# B&R Automation Studio project VPAKRT
Automation Studio 4.0.17.85 SP

## Configuration Simulation

CPU , AutomationRuntime D4.05

### Task classes (Cpu.sw)
```
Cyclic#1 (cycle 2000 us, tolerance 0 us):
  Reject <- Reject.prg
  main <- main.prg
  Entry <- Entry.prg
  CheckRejec <- CheckReject.prg
  Accumulato <- Accumulator.prg
  Camera1 <- Camera1.prg
  Printer <- Printer.prg
  Conveyor <- Conveyor.prg
Cyclic#4 (cycle 1000000 us, tolerance 10000000 us):
  SerialCode <- SerialCodes.prg
  IHM <- IHM.prg
VcDataObjects: Visu <- Visu.dob
Binaries: sysconf, ashwd, asfw, iomap, arconfig
Libraries: CPP, standard, AsHttp, runtime, AsIecCon, astime, FileIO, sys_lib
```

### Hardware
```
PC_any : PC_any v1.1.0.0 (OrderNumber=PC)
  Connector IF3:
    Vnc1
    VncVcObjectName1 = Visu
    VncKeyMappingFile1 = VC\PS2-Keyboard.dis
  SystemTick = 2000
  TaskClassIdleTime = 2000
  Cyclic1Duration = 2000
  Cyclic1Tolerance = 0
  Cyclic1Output = 1
  Cyclic2Duration = 200000
  Cyclic2Tolerance = 10000000
  Cyclic3Duration = 500000
  Cyclic3Tolerance = 10000000
  Cyclic4Duration = 1000000
  Cyclic4Tolerance = 10000000
  Cyclic5Duration = 2000000
  Cyclic5Tolerance = 10000000
  Cyclic6Duration = 3000000
  Cyclic6Tolerance = 12000000
  Cyclic7Duration = 4000000
  Cyclic7Tolerance = 12000000
  Cyclic8Duration = 5000000
  Cyclic8Tolerance = 30000000
  FileDevice1
  FileDeviceName1 = HD0
  FileDevicePath1 = C:\TEMP
```

## Logical view

Binary libraries used (declarations not repeated): standard, AsHttp, runtime, AsIecCon, astime, FileIO, sys_lib

### Global.typ - Global data types
```iecst
(********************************************************************
 * COPYRIGHT -- Pollux
 ********************************************************************
 * File: Global.typ
 * Author: CEDRIC
 * Created: July 16, 2014
 ********************************************************************
 * Global data types of project VPakRT
 ********************************************************************)

TYPE
	Mark : 	STRUCT
		FabricationDate : STRING[20];
		ValidityDate : STRING[20];
		Drug : STRING[20];
		Lot : STRING[20];
		GTIN : STRING[20];
	END_STRUCT;
	status :
		(
		STANDBY,
		ERROR,
		AUTOMATIC,
		MANUAL
		);
	Serial :STRING[20];
	Part : 	STRUCT
		nWidth : UINT;
		nPosition : UINT;
		bRejected : BOOL;
		bResult : BOOL;
		bCamera1 : BOOL;
		bPrinted : BOOL;
		bPresent : BOOL;
		sSerial : Serial;
	END_STRUCT;
	alarm_tower : 	STRUCT
		yellow : BOOL;
		green : BOOL;
		red : BOOL;
	END_STRUCT;
END_TYPE
```

### Global.var - Global variables
```iecst
(********************************************************************
 * COPYRIGHT -- Pollux
 ********************************************************************
 * File: Global.var
 * Author: CEDRIC
 * Created: July 16, 2014
 ********************************************************************
 * Global variables of project VPakRT
 ********************************************************************)
VAR
	gSerialQueue : UDINT := 0; (*Pointer for the queue of serial codes*)
	gConsecutiveRejects : USINT := 5; (*Allowed number of consecutive rejects before stopping*)
END_VAR
VAR RETAIN
	Parts : ARRAY[0..49] OF Part := [50((0))]; (*The FIFO of parts*)
END_VAR
VAR
	doAccumulator : BOOL := FALSE;
	doReject : BOOL := FALSE;
	doCam1TRG : BOOL := FALSE;
	doPrinter : BOOL := FALSE;
	doConveyor : USINT := 0;
	doAlarmTower : alarm_tower := (0);
	diAccumulator : BOOL := FALSE;
	diCheckReject : BOOL := FALSE;
	diCam1RES : BOOL := FALSE;
	diCam1DV : BOOL := FALSE;
	diPrinterReady : BOOL := FALSE;
	diEntry : BOOL := FALSE;
	diEmergency : BOOL := FALSE;
	gHost : STRING[80] := '192.168.0.133'; (*Host server address (default 10.0.0.1)*)
	gOffsetCheckReject : UINT := 400; (*Offset of check reject position*)
	gOffsetReject : UINT := 300; (*Offset of reject position*)
	gOffsetCamera : UINT := 200; (*Offset of camera position*)
	gOffsetPrinter : UINT := 100; (*Offset of printer position*)
	gSystemUUID : STRING[20] := '99dSBT8TwOwfH8wRnGFX';
	gLotNumber : STRING[20] := '123456789';
	gUserUUID : STRING[20] := 'rKsGKLZL9WYUcbvHhipc';
	gMark : Mark := (0); (*The current marking data (GTIN, Lot number, drug number, ...)*)
	gSpeed : UDINT := 0;
	gMoving : USINT := 0; (*Inform if the equipment is moving or not*)
	gMode : status := (0); (*Defines the machine status (manual, automatic, ...)*)
END_VAR
```

### Program Logical/main (ANSIC) - Monitor machine status

#### main.cpp - Implementation code
```cpp
/********************************************************************
 * COPYRIGHT -- Pollux
 ********************************************************************
 * Program: main
 * File: main.cpp
 * Author: CEDRIC
 * Created: July 17, 2014
 ********************************************************************
 * Implementation of program main
 ********************************************************************/

#include <bur/plctypes.h>

#ifdef _DEFAULT_INCLUDES
	#include <AsDefault.h>
#endif
#include <standard.h>

unsigned long bur_heap_size = 0xFFFF; /* Must be added manually */
#include "../CPP/SerialCodes.h"

void _INIT mainInit(void)
{
	gMode	= MANUAL;
	gSerialQueue = (UDINT)createSerialQueue();
}

void _CYCLIC mainCyclic(void)
{
	switch( gMode )
	{
		case MANUAL: // Manual
			gMoving = false;
			doAlarmTower.green	= false;
			doAlarmTower.yellow	= true;
			doAlarmTower.red	= false;
			gMode = STANDBY;
			break;

		case AUTOMATIC:	// Automatic
			gMoving = true;
			doAlarmTower.green	= true;
			doAlarmTower.yellow	= false;
			doAlarmTower.red	= false;
			gMode = STANDBY;
			break;

		case ERROR:	// error
			gMoving = false;
			doAlarmTower.green	= false;
			doAlarmTower.yellow	= false;
			doAlarmTower.red	= true;
			gMode = STANDBY;
			break;

		case STANDBY:	// standby
			break;
	}
}

void _EXIT mainExit(void)
{
	// Release the serial queue
	freeSerialQueue((queue_serial*)gSerialQueue);
}
```

### Program Logical/Entry (ANSIC) - Entry of products

#### Entry.cpp - Implementation code
```cpp
/********************************************************************
 * COPYRIGHT -- Pollux
 ********************************************************************
 * Program: Entry
 * File: Entry.cpp
 * Author: CEDRIC
 * Created: July 17, 2014
 ********************************************************************
 * Implementation of program Entry
 ********************************************************************/

#include <bur/plctypes.h>

#ifdef _DEFAULT_INCLUDES
	#include <AsDefault.h>
#endif

unsigned long bur_heap_size = 0xFFFF; /* Must be added manually */

//#include "File.h"
#include <string.h>
#include "../CPP/Json.h"
#include "../CPP/SerialCodes.h"

int add_part();

void _INIT EntryInit(void)
{
	step	= 0;
}

void _CYCLIC EntryCyclic(void)
{
	switch( step )
	{
		case 10:	// Check size (low)
			if( gSerialQueue == 0 )
				break;
			size = getSerialQueueSize( (queue_serial*)gSerialQueue );
			if( size == 0  )
				gMoving		= false;
			else
			{
				gMoving	= true;
				step	= 20;
			}
			break;

		case 20:	// Read one code
			strcpy( serial_code, popSerialCodeFromQueue( (queue_serial*)gSerialQueue ) );
			step = 30;
			break;

		case 30:	// Wait sensor
			if( diEntry == true )
			{
				position = add_part();
				if( position >= 0 )
					step = 40;
			}
			break;

		case 40:
			if( diEntry == false )
			{
				Parts[position].nWidth = Parts[position].nPosition;
				strcpy( Parts[position].sSerial, serial_code );
				step = 10;
			}
			break;
	}

}

void _EXIT EntryExit(void)
{
}

int part_index( int position )
{
	for( int i=0; i<50; i++ )
		{
		if( Parts[i].bPresent == true )
		{
			if( Parts[i].nPosition == position )
				return i;
		}
	}

	// No position matches
	return -1;
}

int add_part()
{
	for( int i=0; i<50; i++ )
		{
		if( Parts[i].bPresent == false )
		{
			Parts[i].bPresent = true;
			Parts[i].nPosition	= 0;
			Parts[i].nWidth		= 0;
			Parts[i].bPrinted	= false;
			Parts[i].bCamera1	= false;
			Parts[i].bRejected	= false;
			Parts[i].bResult	= false;
			return i;
		}
	}

	// No position found!!
	return -1;
}
```

#### Entry.var - Local variables
```iecst
(********************************************************************
 * COPYRIGHT -- Pollux
 ********************************************************************
 * Program: Entry
 * File: Entry.var
 * Author: CEDRIC
 * Created: July 17, 2014
 ********************************************************************
 * Local variables of program Entry
 ********************************************************************)
VAR
	serial_code : Serial := (0);
	position : INT := 0;
	size : INT := 0;
	step : INT := 0;
END_VAR
```

#### File.h
```c
/********************************************************************
 * COPYRIGHT -- Pollux
 ********************************************************************
 * Program: Entry
 * File: File.h
 * Author: CEDRIC
 * Created: July 24, 2014
 *******************************************************************/

#include <bur/plctypes.h>
#include <fileio.h>
#include <string.h>

class File
{
	private:
	char m_Device[80];
	char m_Filename[80];
	UDINT m_wId;
	UINT m_uErrorCode;
	UINT m_uStatus;
	BOOL m_bError;
	FileOpen_typ m_fopen;
	FileClose_typ m_fclose;
	FileCreate_typ m_fcreate;
	FileRead_typ m_fread;
	FileWrite_typ m_fwrite;
	FileInfo_typ m_info;
	fiFILE_INFO m_tinfo;
	int m_step;

	public:
	File( char *Device, char *Filename );
	~File();

	INT close();
	INT create();
	INT get_size( UDINT* size );
	INT open();
	INT read( UDINT buffer, UDINT length, UDINT offset );
	INT read_info();
	INT write( UDINT buffer, UDINT length, UDINT offset );
};
```

#### File.cpp
```cpp
/********************************************************************
 * COPYRIGHT -- Pollux
 ********************************************************************
 * Program: Entry
 * File: File.cpp
 * Author: CEDRIC
 * Created: July 24, 2014
 *******************************************************************/

#include <bur/plctypes.h>
#ifdef _DEFAULT_INCLUDES
	#include <AsDefault.h>
#endif

#include "File.h"

File::File( char *Device, char *Filename )
{
	m_bError		= false;
	m_uErrorCode	= 0;
	m_wId			= 0;
	m_uStatus		= 0;
	m_step			= 10;
	memset( &m_fopen, 0, sizeof(FileOpen_typ) );
	memset( &m_fcreate, 0, sizeof(FileCreate_typ) );
	memset( &m_fread, 0, sizeof(FileRead_typ) );
	memset( &m_fwrite, 0, sizeof(FileWrite_typ) );
	memset( &m_fclose, 0, sizeof(FileClose_typ) );
	strncpy( m_Device, Device, 80 );
	strncpy( m_Filename, Filename, 80 );
}

File::~File()
{
	this->close();
}

INT File::close()
{
	m_fclose.enable	= 1;
	m_fclose.ident	= m_wId;
	FileClose( &m_fclose );

	m_uStatus	= m_fclose.status;

	switch( m_uStatus )
	{
		case 0:		// Ok
			m_bError	= false;
			return 1;
			break;

		case 65535:	// Busy
			return 0;
			break;

		case 20799:	//
			m_bError	= true;
			m_uErrorCode	= FileIoGetSysError();
			return -2;
			break;

		default:	// Other errors
			m_bError	= true;
			return -3;
			break;
	}
}

INT File::create()
{
	m_fcreate.enable    = 1;
	m_fcreate.pDevice = (UDINT)m_Device;
	m_fcreate.pFile   = (UDINT)m_Filename;
	/* Call FUB */
	FileCreate(&m_fcreate);

	/* Get output information of FBK */
	m_wId		= m_fcreate.ident;
	m_uStatus	= m_fcreate.status;

	switch( m_uStatus )
	{
		case 0:		// Ok
			return 1;
			break;

		case 65535:	// Busy
			return 0;
			break;

		case 20799:	// File IO error
			m_bError		= true;
			m_uErrorCode	= FileIoGetSysError();
			return -1;
			break;

		default:	// Other errors
			m_bError	= true;
			return -3;
			break;
	}
}

INT File::get_size( UDINT *size )
{
	int return_code = 0;

	switch( m_step )
	{
		case 10:	// Get file information
			switch( this->read_info() )
			{
				case 0:	// Busy
					break;

				case 1:	// Ok
					m_step = 20;
					break;

				default:
					return_code = -3;
					break;
			}
			break;

		case 20:	// Get file size
			*size = m_tinfo.size;
			return_code = 1;
			m_step = 10;
			break;
	}

	return return_code;
}

INT File::open()
{
	m_fopen.enable    = 1;
	m_fopen.pDevice = (UDINT)m_Device;
	m_fopen.pFile   = (UDINT)m_Filename;
	m_fopen.mode	= FILE_RW;
	/* Call FUB */
	FileOpen(&m_fopen);

	/* Get output information of FBK */
	m_wId		= m_fopen.ident;
	m_uStatus	= m_fopen.status;

	/* Status OK? */
	switch( m_uStatus )
	{
		case 0:	// OK
			return 1;
			break;

		case 65535:	// Busy
			return 0;
			break;

		case 20708:	// Not exist
			m_bError	= true;
			return -1;
			break;

		case 20799:	// File IO error
			m_bError		= true;
			m_uErrorCode	= FileIoGetSysError();
			return -2;
			break;

		default:	// Other errors
			m_bError	= true;
			return -3;
			break;
	}
}

INT File::read( UDINT buffer, UDINT length, UDINT offset )
{
	m_fread.enable      = 1;
	m_fread.ident     = m_wId;
	m_fread.offset    = offset;
	m_fread.pDest     = buffer;
	m_fread.len       = length;
	/* Call FBK */
	FileRead(&m_fread);
	/* Get status */
	m_uStatus = m_fread.status;

	/* Verify status */
	switch( m_uStatus )
	{
		case 0:		// Ok
			return 1;
			break;

		case 65535:	// Busy
			return 0;
			break;

		case 20799:	// File IO error
			m_bError		= true;
			m_uErrorCode	= FileIoGetSysError();
			return -1;
			break;

		default:	// Other cases
			m_bError	= true;
			return -3;
			break;
	}
}

INT File::read_info()
{
	m_info.enable	= 1;
	m_info.pDevice	= (UDINT)m_Device;
	m_info.pName	= (UDINT)m_Filename;
	m_info.pInfo	= (UDINT)&m_tinfo;

	FileInfo( &m_info );

	switch( m_info.status )
	{
		case 0:		// Ok
			return 1;
			break;

		case 65535:	// Busy
			return 0;
			break;

		default:	// All errors
			return -3;
			break;
	}
}

INT File::write( UDINT buffer, UDINT length, UDINT offset )
{
	m_fwrite.enable     = 1;
	m_fwrite.ident    = m_wId;
	m_fwrite.offset   = offset;
	m_fwrite.pSrc     = buffer;
	m_fwrite.len      = length;

	/* Call FBK */
	FileWrite(&m_fwrite);
	/* Get status */
	m_uStatus = m_fwrite.status;

	switch( m_uStatus )
	{
		case 0:		// Ok
			return 1;
			break;

		case 65535:	// Busy
			return 0;
			break;

		case 20799:	// File IO error
			m_bError		= true;
			m_uErrorCode	= FileIoGetSysError();
			return -2;
			break;

		default:	// Other errors
			m_bError	= true;
			return -3;
			break;
	}
}
```

### Program Logical/Conveyor (ANSIC) - Machine Conveyor

#### Conveyor.cpp - Implementation code
```cpp
/********************************************************************
 * COPYRIGHT -- Pollux
 ********************************************************************
 * Program: Conveyor
 * File: Conveyor.cpp
 * Author: CEDRIC
 * Created: July 16, 2014
 ********************************************************************
 * Implementation of program Conveyor
 ********************************************************************/

#include <bur/plctypes.h>

#ifdef _DEFAULT_INCLUDES
	#include <AsDefault.h>
#endif

unsigned long bur_heap_size = 0xFFFF; /* Must be added manually */

#include "../CPP/Timer.h"

void shift_parts();

Timer* pTimer;
void _INIT ConveyorInit(void)
{
	step = 10;
	pTimer = new Timer(1);
}

void _CYCLIC ConveyorCyclic(void)
{
	switch( step )
	{
		case 10:	// Check if movement allowed
			if( gMoving == true )
				step = 20;
			break;

		case 20:	// Set output to 1
			doConveyor = true;
			pTimer->start();
			step = 30;
			break;

		case 30:	// Wait timer
			pTimer->cyclic();
			if( pTimer->getOutput() == true )
				step = 40;
			break;

		case 40:	// Set output to 0
			doConveyor = false;
			pTimer->stop();
			step = 10;
			// Shift register
			shift_parts();
			break;
	}
}

void _EXIT ConveyorExit(void)
{
	delete pTimer;
}

void shift_parts()
{
	for( int i=0; i<50; i++)
		{
		if( Parts[i].bPresent == true )
		{
			Parts[i].nPosition++;
		}
	}
}
```

#### Conveyor.var - Local variables
```iecst
(********************************************************************
 * COPYRIGHT -- Pollux
 ********************************************************************
 * Program: Conveyor
 * File: Conveyor.var
 * Author: CEDRIC
 * Created: July 16, 2014
 ********************************************************************
 * Local variables of program Conveyor
 ********************************************************************)
VAR
	step : USINT := 0;
END_VAR
```

### Program Logical/Printer (ANSIC) - Printer management

#### Printer.cpp - Implementation code
```cpp
/********************************************************************
 * COPYRIGHT -- Pollux
 ********************************************************************
 * Program: Printer
 * File: Printer.cpp
 * Author: CEDRIC
 * Created: July 17, 2014
 ********************************************************************
 * Implementation of program Printer
 ********************************************************************/

#include <bur/plctypes.h>

#ifdef _DEFAULT_INCLUDES
	#include <AsDefault.h>
#endif
unsigned long bur_heap_size = 0xFFFF; /* Must be added manually */

#include "../CPP/Timer.h"

Timer *timerPrinter;
void _INIT PrinterInit(void)
{
	step			= 10;
	timerPrinter	= new Timer(100);
	position		= -1;
}

void _CYCLIC PrinterCyclic(void)
{
	switch( step )
	{
		case 10:	// Wait ACK to print
			for( int i=0; i<50; i++ )
			{
				if( Parts[i].bPresent == true && Parts[i].bPrinted == false )
				{
					if( Parts[i].nPosition == gOffsetPrinter )
					{
						position = i;
						step = 20;
					}
				}
			}
			break;

		case 20:	// Start printing
			doPrinter = true;
			timerPrinter->start();
			step = 30;
			break;

		case 30:
			timerPrinter->cyclic();
			if( timerPrinter->getOutput() == true )
			{
				doPrinter = false;
				step = 10;
				Parts[position].bPrinted = true;
			}
			break;
	}
}

void _EXIT PrinterExit(void)
{
	delete timerPrinter;
}
```

#### Printer.var - Local variables
```iecst
(********************************************************************
 * COPYRIGHT -- Pollux
 ********************************************************************
 * Program: Printer
 * File: Printer.var
 * Author: CEDRIC
 * Created: July 17, 2014
 ********************************************************************
 * Local variables of program Printer
 ********************************************************************)
VAR
	position : INT := 0;
	step : USINT := 0;
END_VAR
```

### Program Logical/Camera1 (ANSIC) - Camera 1 management

#### Camera1.cpp - Implementation code
```cpp
/********************************************************************
 * COPYRIGHT -- Pollux
 ********************************************************************
 * Program: Camera1
 * File: Camera1.cpp
 * Author: CEDRIC
 * Created: July 17, 2014
 ********************************************************************
 * Implementation of program Camera1
 ********************************************************************/

#include <bur/plctypes.h>

#ifdef _DEFAULT_INCLUDES
	#include <AsDefault.h>
#endif
unsigned long bur_heap_size = 0xFFFF; /* Must be added manually */

#include <string.h>
#include "../CPP/Timer.h"
#include "../CPP/Json.h"

#define	URL_TEST			"~cedriccraze/vpackRT/services/index.php?user_UUID=%s&system_UUID=%s&lot_number=%s&quantity=%d"
#define	URL_UPDATE_STATUS	"~cedriccraze/vpackRT/services/update_ium_status.php?user_UUID=%s&system_UUID=%s&serial=%s&status=%d"

#define	STATUS_VALID		2
#define	STATUS_NOT_VALID	3

Timer* timer;
void _INIT Camera1Init(void)
{
	step		= 10;
	step_http	= 0;
	timer		= new Timer(100);
	position	= -1;

	// HTTP Client comunication
	client.enable			= false;
	client.abort			= false;
	client.send				= false;
	client.hostPort			= 0;
	client.method			= httpMETHOD_GET;
	client.option			= httpOPTION_HTTP_11;
	client.pHost			= (long unsigned int)gHost;
	client.pRequestData		= 0;
	client.pRequestHeader	= 0;
	client.pResponseData	= (long unsigned int)response;
	client.pResponseHeader	= 0;
	client.pStatistics		= 0;
	client.pStruct			= 0;
	client.pUri				= (long unsigned int)url;
	client.requestDataLen	= 0;
	client.responseDataSize	= sizeof(response);
}

void _CYCLIC Camera1Cyclic(void)
{
	switch( step )
	{
		case 10:	// Send code to printer
			for( int i=0; i<50; i++ )
				{
				if( Parts[i].bPresent == true && Parts[i].bCamera1 == false )
				{
					if( Parts[i].nPosition == gOffsetCamera )
					{
						position = i;
						step = 20;
					}
				}
			}
			break;

		case 20:	// Start trigger
			doCam1TRG = true;
			timer->start();
			step = 30;
			break;

		case 30:	// Stop trigger
			timer->cyclic();
			if( timer->getOutput() == true )
			{
				doCam1TRG = false;
				step = 40;
			}
			break;

		case 40:	// Wait DV
			if( diCam1DV == true )
			{
				Parts[position].bResult		= diCam1RES;
				Parts[position].bCamera1	= true;

				step = 50;
			}
			break;

		case 50:	// Wait HTTP
			if( step_http == 0 )
			{
				// Update server
				step_http = 10;
				// Copy data
				memcpy( &part, &Parts[position], sizeof(Part) );

				step = 10;
			}
			else	// OVERRUN !!!
			{
				gMoving	= false;
				gMode	= ERROR;
				step	= 999;
			}
			break;
	}

	// HTTP Communication
	httpClient(&client);
	switch( step_http )
	{
		case 10:	// Start HTTP
			memset( response, 0, sizeof(response) );
			sprintf( url, URL_UPDATE_STATUS, gUserUUID, gSystemUUID, part.sSerial, part.bResult == true ? STATUS_VALID : STATUS_NOT_VALID  );
			client.enable	= true;
			client.send		= true;
			step_http		= 20;
			break;

		case 20:	// Wait HTTP processing
			switch( client.status )
			{
				case 0:		// Ok
					client.send	= false;
					step_http		= 30;
					break;

				case 65535:	// BUSY
					break;

				default:	// Error
					step_http	= 999;
					break;
			}
			break;

		case 30:	// Wait response
			if( strlen(response) > 0 )
				step_http = 40;
			break;

		case 40:	// JSON decodification
			{
				JsonError error;
				JsonObject* root = (JsonObject*)json_decode( response, &error );
				if( root == NULL || root->get_type() != kJSON_OBJECT )
				{
					step_http = 999;
					break;
				}

				JsonValue* value = (JsonValue*)root->key_value("result");
				if( value == NULL || strcmp( value->string_value(), "NOK" ) == 0 )
				{
					step_http = 998;
					break;
				}
				if( strcmp( value->string_value(), "OK" ) != 0 )
				{
					step_http = 997;
					break;
				}

				// End communication
				step_http	= 0;
			}
			break;
	}
}

void _EXIT Camera1Exit(void)
{
	delete timer;
}
```

#### Camera1.var - Local variables
```iecst
(********************************************************************
 * COPYRIGHT -- Pollux
 ********************************************************************
 * Program: Camera1
 * File: Camera1.var
 * Author: CEDRIC
 * Created: July 17, 2014
 ********************************************************************
 * Local variables of program Camera1
 ********************************************************************)
VAR
	step_http : INT := 0;
	part : Part := (0);
	url : STRING[500] := '~cedriccraze/vpackRT/services/index.php';
	response : STRING[100000];
	client : httpClient := (0);
	position : INT := 0;
	step : INT := 0;
END_VAR
```

### Program Logical/Reject (ANSIC) - Reject management

#### Reject.cpp - Implementation code
```cpp
/********************************************************************
 * COPYRIGHT -- Pollux
 ********************************************************************
 * Program: Reject
 * File: Reject.cpp
 * Author: CEDRIC
 * Created: July 17, 2014
 ********************************************************************
 * Implementation of program Reject
 ********************************************************************/

#include <bur/plctypes.h>

#ifdef _DEFAULT_INCLUDES
	#include <AsDefault.h>
#endif
unsigned long bur_heap_size = 0xFFFF; /* Must be added manually */

#include "../CPP/Timer.h"

Timer* timer;
void _INIT RejectInit(void)
{
	step		= 10;
	timer		= new Timer(50);
	position	= -1;
}

void _CYCLIC RejectCyclic(void)
{
	switch( step )
	{
		case 10:
			for( int i=0; i<50; i++ )
				{
				if( Parts[i].bPresent == true && Parts[i].bResult == false )
				{
					if( Parts[i].nPosition == gOffsetReject )
					{
						position = i;
						step = 20;
					}
				}
			}
			break;

		case 20:	// Start trigger
			doReject = true;
			consecutive_rejects++;
			timer->start();
			step = 30;
			break;

		case 30:	// Stop trigger
			timer->cyclic();
			if( timer->getOutput() == true )
			{
				doReject = false;
				if( consecutive_rejects == gConsecutiveRejects )
					step = 40;
				else
					step = 10;
			}
			break;

		case 40:	// Consecutive rejects
			gMoving	= false;
			gMode	= ERROR;
			// TODO
			// - Go to specific screen
			// - Allow user to stop/pause/continue
			break;
	}
}

void _EXIT RejectExit(void)
{
	delete timer;
}
```

#### Reject.var - Local variables
```iecst
(********************************************************************
 * COPYRIGHT -- Pollux
 ********************************************************************
 * Program: Reject
 * File: Reject.var
 * Author: CEDRIC
 * Created: July 17, 2014
 ********************************************************************
 * Local variables of program Reject
 ********************************************************************)
VAR
	consecutive_rejects : USINT := 0;
	position : INT := 0;
	step : USINT := 0;
END_VAR
```

### Program Logical/CheckReject (ANSIC) - Check reject management

#### CheckReject.cpp - Implementation code
```cpp
/********************************************************************
 * COPYRIGHT -- Pollux
 ********************************************************************
 * Program: CheckReject
 * File: CheckReject.cpp
 * Author: CEDRIC
 * Created: July 17, 2014
 ********************************************************************
 * Implementation of program CheckReject
 ********************************************************************/

#include <bur/plctypes.h>

#ifdef _DEFAULT_INCLUDES
	#include <AsDefault.h>
#endif
unsigned long bur_heap_size = 0xFFFF; /* Must be added manually */

#include "../CPP/Timer.h"

Timer* timer;
void _INIT CheckRejectInit(void)
{
	step		= 10;
	position	= -1;
}

void _CYCLIC CheckRejectCyclic(void)
{
	switch( step )
	{
		case 10:
			for( int i=0; i<50; i++ )
			{
				if( Parts[i].bPresent == true && Parts[i].bResult == false )
				{
					if( Parts[i].nPosition == gOffsetCheckReject )
					{
						position = i;
						step = 20;
					}
				}
			}
			break;

		case 20:
			if( diCheckReject == true )
			{
				gMode = ERROR;
			}
			else
				step = 10;
			break;
	}
}

void _EXIT CheckRejectExit(void)
{
	/* TODO: Add code here */
}
```

#### CheckReject.var - Local variables
```iecst
(********************************************************************
 * COPYRIGHT -- Pollux
 ********************************************************************
 * Program: CheckReject
 * File: CheckReject.var
 * Author: CEDRIC
 * Created: July 17, 2014
 ********************************************************************
 * Local variables of program CheckReject
 ********************************************************************)
VAR
	position : INT := 0;
	step : USINT := 0;
END_VAR
```

### Program Logical/Accumulator (ANSIC) - Accumulator management

#### Accumulator.cpp - Implementation code
```cpp
/********************************************************************
 * COPYRIGHT -- Pollux
 ********************************************************************
 * Program: Accumulator
 * File: Accumulator.cpp
 * Author: CEDRIC
 * Created: July 22, 2014
 ********************************************************************
 * Implementation of program Accumulator
 ********************************************************************/

#include <bur/plctypes.h>

#ifdef _DEFAULT_INCLUDES
	#include <AsDefault.h>
#endif

unsigned long bur_heap_size = 0xFFFF; /* Must be added manually */

#include "../CPP/Timer.h"

Timer* timer;
void _INIT AccumulatorInit(void)
{
	step = 10;
	timer = new Timer(1000);
}

void _CYCLIC AccumulatorCyclic(void)
{
	switch( step )
	{
		case 10:	// WAIT accumulator == TRUE
			if( diAccumulator == true )
			{
				timer->start();
				step = 20;
			}
			else
			{
				if( gMode != AUTOMATIC )
				{
					doAccumulator = true;
					step = 40;
				}
			}
			break;

		case 20:	// WAIT timer
			timer->cyclic();
			if( timer->getOutput() == true )
			{
				gMoving = false;
				doAccumulator = true;
				step = 30;
			}
			else 	// WAIT reset accumulator?
			{
				if( diAccumulator == false )
				{
					timer->stop();
					step = 10;
				}
			}
			break;

		case 30:	// WAIT accumulator = FALSE
			if( diAccumulator == false )
			{
				gMoving = true;
				doAccumulator = false;
				step = 10;
			}
			break;

		case 40:	// Not in automatic
			if( gMode == AUTOMATIC )
			{
				doAccumulator = false;
				step = 10;
			}
			break;
	}
}

void _EXIT AccumulatorExit(void)
{
	delete timer;
}
```

#### Accumulator.var - Local variables
```iecst
(********************************************************************
 * COPYRIGHT -- Pollux
 ********************************************************************
 * Program: Accumulator
 * File: Accumulator.var
 * Author: CEDRIC
 * Created: July 22, 2014
 ********************************************************************
 * Local variables of program Accumulator
 ********************************************************************)
VAR
	step : USINT := 0;
END_VAR
```

### Program Logical/SerialCodes (ANSIC) - Serial Codes queue management

#### SerialCodes.cpp - Implementation code
```cpp
/********************************************************************
 * COPYRIGHT -- Pollux
 ********************************************************************
 * Program: SerialCodes
 * File: SerialCodes.cpp
 * Author: CEDRIC
 * Created: August 01, 2014
 ********************************************************************
 * Implementation of program SerialCodes
 ********************************************************************/

#include <bur/plctypes.h>

#ifdef _DEFAULT_INCLUDES
	#include <AsDefault.h>
#endif

unsigned long bur_heap_size = 0xFFFF; /* Must be added manually */

#include <string.h>
#include "../CPP/Json.h"
#include "../CPP/SerialCodes.h"

#define	URL_TEST			"~cedriccraze/vpackRT/services/index.php?user_UUID=%s&system_UUID=%s&lot_number=%s&quantity=%d"
#define	URL_REQUEST_SERIAL	"~cedriccraze/vpackRT/services/request_iums.php?user_UUID=%s&system_UUID=%s&lot_number=%s&quantity=%d"

void _INIT SerialCodesInit(void)
{
	step	= 0;

	// HTTP Client comunication
	client.enable			= false;
	client.abort			= false;
	client.send				= false;
	client.hostPort			= 0;
	client.method			= httpMETHOD_GET;
	client.option			= httpOPTION_HTTP_11;
	client.pHost			= (long unsigned int)gHost;
	client.pRequestData		= 0;
	client.pRequestHeader	= 0;
	client.pResponseData	= (long unsigned int)response;
	client.pResponseHeader	= 0;
	client.pStatistics		= 0;
	client.pStruct			= 0;
	client.pUri				= (long unsigned int)url_request_serial;
	client.requestDataLen	= 0;
	client.responseDataSize	= sizeof(response);
}

void _CYCLIC SerialCodesCyclic(void)
{
	// HTTP Communication
	httpClient(&client);
	switch( step )
	{
		case 10:	// Send request
			if( gSerialQueue == 0 )
				break;
			size	= getSerialQueueSize((queue_serial*)gSerialQueue);
			if( size < 50 )
			{
				memset( response, 0, sizeof(response) );
				sprintf( url_request_serial, URL_REQUEST_SERIAL, gUserUUID, gSystemUUID, gLotNumber, 400-getSerialQueueSize((queue_serial*)gSerialQueue) );
				client.enable	= true;
				client.send		= true;
				step			= 20;
			}
			break;

		case 20:	// Wait communication
			switch( client.status )
			{
				case 0:		// Ok
					client.send = false;
					step		= 30;
					break;

				case 65535:	// Busy
					break;

				case 65534:	// Enable
					break;

				default:	// Error
					client.send	= false;
					step		= 999;
					break;
			}
			break;

		case 30:	// Wait response
			if( strlen(response) > 0 )
				step = 40;
			break;

		case 40:	// JSON
			{
				JsonError error;
				JsonObject* root = (JsonObject*)json_decode( response, &error );
				if( root == NULL || root->get_type() != kJSON_OBJECT )
				{
					step = 999;
					break;
				}

				JsonValue* value = (JsonValue*)root->key_value("result");
				if( value == NULL || strcmp( value->string_value(), "NOK" ) == 0 )
				{
					step = 998;
					break;
				}
				if( strcmp( value->string_value(), "OK" ) != 0 )
				{
					step = 997;
					break;
				}

				JsonArray* codes = (JsonArray*)root->key_value("codes");
				if( codes == NULL || codes->get_type() != kJSON_ARRAY )
				{
					step = 996;
					break;
				}
				for( int i=0; i<codes->getsize(); i++ )
					{
					value = (JsonValue*)codes->get_at(i);
					if( value == NULL || value->get_type() != kJSON_STRING)
					{
						step = 995;
						break;
					}

					pushSerialCodeToQueue((queue_serial*)gSerialQueue, value->string_value() );
				}

				if( step < 900 )
					step = 10;

				// Free memory
				delete root;
			}
			break;

		default:
			gMode	= ERROR;
			gMoving	= false;
			break;
	}
}

void _EXIT SerialCodesExit(void)
{
	client.enable	= false;
	client.send		= false;
}
```

#### SerialCodes.var - Local variables
```iecst
(********************************************************************
 * COPYRIGHT -- Pollux
 ********************************************************************
 * Program: SerialCodes
 * File: SerialCodes.var
 * Author: CEDRIC
 * Created: August 01, 2014
 ********************************************************************
 * Local variables of program SerialCodes
 ********************************************************************)
VAR
	size : INT := 0;
	url_request_serial : STRING[500] := '~cedriccraze/vpackRT/services/request_ium.php';
	response : STRING[100000];
	client : httpClient := (0);
	step : INT := 0;
END_VAR
```

- Visualisation Logical/Visu (not shown)

### Program Logical/IHM (ANSIC) - Gerenciamento IHM

#### IHM.cpp - Implementation code
```cpp
/********************************************************************
 * COPYRIGHT -- Pollux
 ********************************************************************
 * Program: IHM
 * File: IHM.cpp
 * Author: CEDRIC
 * Created: August 13, 2014
 ********************************************************************
 * Implementation of program IHM
 ********************************************************************/

#include <bur/plctypes.h>

#ifdef _DEFAULT_INCLUDES
	#include <AsDefault.h>
#endif

unsigned long bur_heap_size = 0xFFFF; /* Must be added manually */

#include <string.h>
#include "../CPP/Json.h"
#include "../CPP/SerialCodes.h"

void _INIT IHMInit(void)
{
	step	= 10;
	nActivePage	= 10;

	// HTTP Client comunication
	client.enable			= false;
	client.abort			= false;
	client.send				= false;
	client.hostPort			= 0;
	client.method			= httpMETHOD_GET;
	client.option			= httpOPTION_HTTP_11;
	client.pHost			= (long unsigned int)gHost;
	client.pRequestData		= 0;
	client.pRequestHeader	= 0;
	client.pResponseData	= (long unsigned int)response;
	client.pResponseHeader	= 0;
	client.pStatistics		= 0;
	client.pStruct			= 0;
	client.pUri				= (long unsigned int)url_request_serial;
	client.requestDataLen	= 0;
	client.responseDataSize	= sizeof(response);
}

void _CYCLIC IHMCyclic(void)
{
	httpClient(&client);

	switch( step )
	{
		case 10:	// Check system UUID
			if( strlen( gSystemUUID ) < 20 )
				step = 20;
			else
				step = 100;
			break;

		case 20:	// Send message to server
			memset( response, 0, sizeof(response));
			client.enable	= true;
			client.send		= true;
			step			= 30;
			break;

		case 30:	// Wait answer
			switch( client.status )
			{
				case 0:	// Ok
					client.send	= false;
					step		= 40;
					break;

				case 65535:	// Busy
					break;

				case 65534:	// Enable missing
					break;

				default:	// Error
					break;
			}
			break;

		case 40:	// Wait response
			if( strlen(response) > 0 )
			{
				bServerCom	= true;
				step		= 50;
			}
			break;
	}
}

void _EXIT IHMExit(void)
{
	/* TODO: Add code here */
}
```

#### IHM.var - Local variables
```iecst
(********************************************************************
 * COPYRIGHT -- Pollux
 ********************************************************************
 * Program: IHM
 * File: IHM.var
 * Author: CEDRIC
 * Created: August 13, 2014
 ********************************************************************
 * Local variables of program IHM
 ********************************************************************)
VAR
	nActivePage : UDINT := 0;
	bServerCom : BOOL := FALSE;
	response : STRING[100000];
	url_request_serial : STRING[500] := '~cedriccraze/vpackRT/services/info.php';
	client : httpClient := (0);
	step : UDINT := 0;
END_VAR
```

### Library Logical/CPP (ANSIC) - CPP Library

#### Timer.h
```c
/********************************************************************
 * COPYRIGHT -- Pollux
 ********************************************************************
 * Library: CPP
 * File: Timer.h
 * Author: CEDRIC
 * Created: July 17, 2014
 *******************************************************************/

#include <bur/plctypes.h>
#include <standard.h>
class Timer
{
	private:
	TON_typ fubTON;
	bool started;

	public:
	Timer();
	Timer( signed long time );
	~Timer();

	void cyclic();
	signed long getElapsedTime();
	bool getOutput();
	bool isStarted() const { return this->started; }
	void setTime( signed long time );
	void start();
	void stop();
};
```

#### Timer.cpp
```cpp
/********************************************************************
 * COPYRIGHT -- Pollux
 ********************************************************************
 * Library: CPP
 * File: Timer.cpp
 * Author: CEDRIC
 * Created: July 17, 2014
 *******************************************************************/

#include <bur/plctypes.h>

#include <string.h>
#include "Timer.h"

Timer::Timer()
{
	memset( &this->fubTON, 0, sizeof(this->fubTON) );
	this->started = false;
}

Timer::Timer( signed long time )
{
	memset( &this->fubTON, 0, sizeof(this->fubTON) );
	this->started = false;
	this->setTime( time );
}

Timer::~Timer()
{
}

void Timer::cyclic()
{
	TON(&this->fubTON);
}

signed long Timer::getElapsedTime()
{
	return this->fubTON.ET;
}

bool Timer::getOutput()
{
	return this->fubTON.Q;
}

void Timer::setTime( signed long time )
{
	this->fubTON.PT = time;
}

void Timer::start()
{
	this->fubTON.IN = true;
	this->started = true;
}

void Timer::stop()
{
	this->fubTON.IN = false;
	this->started = false;
}
```

#### Json.h
```c
/********************************************************************
 * COPYRIGHT -- Pollux
 ********************************************************************
 * Library: CPP
 * File: Json.h
 * Author: CEDRIC
 * Created: July 30, 2014
 *******************************************************************/

#ifndef __JSON__
#define __JSON__

#include <bur/plctypes.h>
#include <vector>
#include <string>
#include <map>

using namespace std;

typedef enum
{
	kJSON_ERR_NO_ERROR,
	kJSON_ERR_STRING,		// Missing "
	kJSON_ERR_COLON,		// Missing :
	kJSON_ERR_OBJECT,		// Missing , or }
	kJSON_ERR_ARRAY,		// Missing , or ]
	kJSON_ERR_PARSE_VALUE,	// Syntax error while parsing value
	kJSON_ERR_NO_DATA,		// No data found
}JSON_ERROR;

class JsonError
{
	private:
	string m_sMsg;
	JSON_ERROR m_nCode;
	int m_nPosition;

	public:
	JsonError();

	const char *get_error_string() { return this->m_sMsg.c_str(); }
	JSON_ERROR get_error_code() { return this->m_nCode; }
	int get_position() { return this->m_nPosition; }
	void set_error_code( JSON_ERROR nCode, int position );
};

/* types */
typedef enum {
	kJSON_OBJECT,
	kJSON_ARRAY,
	kJSON_STRING,
	kJSON_INTEGER,
	kJSON_REAL,
	kJSON_TRUE,
	kJSON_FALSE,
	kJSON_NULL
} JSON_TYPE;

class Json
{
	private:
	JSON_TYPE m_type;
	protected:
	JsonError* m_error;

	protected:
	void set_type( JSON_TYPE type ) { m_type = type; };
	string parse_string( string* s, unsigned int* position, char* chars=NULL );
	Json* parse_value( string* s, unsigned int* position );
	public:
	Json( JsonError* error, JSON_TYPE type );
	virtual ~Json();

	virtual void free();
	JSON_TYPE get_type() { return m_type; };
	virtual Json* parse( string* s, unsigned int* position ) { return NULL; };
};

class JsonValue : public Json
{
	private:
	string m_string;

	protected:
	void set_string( string value );
	public:
	JsonValue( JsonError* error, JSON_TYPE type, string value );
	virtual ~JsonValue();

	void free();
	const char* string_value() { return this->m_string.c_str(); }
	int int_value() { return atoi(this->m_string.c_str()); };
	double float_value() { return atof(this->m_string.c_str()); }
	bool bool_value() { if( Json::get_type() == kJSON_TRUE ) return true; else return false; }
};

class JsonObject : public Json
{
	private:
	map<string,Json*> m_keys;

	public:
	JsonObject( JsonError* error );
	virtual ~JsonObject();

	void free();
	Json* parse( string* s, unsigned int* position );
	Json* key_value( string key );
};

class JsonArray : public Json
{
	private:
	vector<Json*> m_values;

	public:
	JsonArray( JsonError* error );
	virtual ~JsonArray();

	void free();
	Json* parse( string* s, unsigned int* position );
	Json* get_at( int index );
	int getsize() { return this->m_values.size(); }
};

Json* json_decode( char* string, JsonError* error );

#endif
```

#### Json.cpp
```cpp
/********************************************************************
 * COPYRIGHT -- Pollux
 ********************************************************************
 * Library: CPP
 * File: Json.cpp
 * Author: CEDRIC
 * Created: July 30, 2014
 *******************************************************************/

#include <bur/plctypes.h>
#include "Json.h"

/*
 * Json class
 *
	*/
Json::Json( JsonError* error, JSON_TYPE type)
{
	this->m_type = type;
	this->m_error = error;
}

Json::~Json()
{
	this->free();
}

void Json::free()
{
}

string Json::parse_string( string* s, unsigned int* position, char* chars/*=NULL*/ )
{
	unsigned int	start	= string::npos;
	unsigned int	end		= string::npos;
	string			str;

	if( chars == NULL )
	{
		// Find first "
		start	= s->find('"', *position);
		if( start != string::npos )
		{
			start++;
			(*position)++;

			// Find second "
			end = s->find( '"', start );
		}
	}
	else
	{
		start	= *position;
		end		= s->find_first_of(chars,*position);
	}

	if( start == string::npos || end == string::npos )
		return str;

	// Build string
	(*position) = end+1;
	int length	= end-start;
	str = s->substr( start, length );
	return str;
}

Json* Json::parse_value( string* s, unsigned int* position )
{
	Json* obj		= NULL;
	bool bParsing	= true;
	string str;
	do
	{
		switch( s->at((*position)) )
		{
			case ' ':	// Do not consider spaces
				break;

			case '"':	// String
				str = this->parse_string(s, position);
				if( str.empty() )
				{
					this->m_error->set_error_code(kJSON_ERR_STRING, *position);
					return NULL;
				}
				obj = new JsonValue(this->m_error,kJSON_STRING, str );
				bParsing	= false;
				break;

			case '{':	// Object
				obj	= new JsonObject(this->m_error);
				(*position)++;
				if( obj->parse(s,position) == NULL )
					return NULL;
				bParsing	= false;
				break;

			case '[':	// Array
				obj = new JsonArray(this->m_error);
				(*position)++;
				if( obj->parse(s,position) == NULL )
					return NULL;
				bParsing = false;
				break;

			case '-':	// Number
			case '+':
			case '.':
			case '0':
			case '1':
			case '2':
			case '3':
			case '4':
			case '5':
			case '6':
			case '7':
			case '8':
			case '9':
			case 'f':	// false
			case 't':	// true
				str = this->parse_string(s,position, ",}");
				if( str.empty() )
				{
					this->m_error->set_error_code(kJSON_ERR_STRING,*position);
					return NULL;
				}
				obj = new JsonValue(this->m_error, kJSON_NULL, str );
				bParsing = false;
				// Decrease index
				(*position)--;
				break;

			case ',':	// Syntax Error
			case ']':
			case '}':
				this->m_error->set_error_code(kJSON_ERR_PARSE_VALUE, *position );
				return NULL;
				break;
		}
	}
	while( bParsing == true && (*position)++ < s->length() );

	return obj;
}

/*
* JsonValue class
*
*/
JsonValue::JsonValue( JsonError* error, JSON_TYPE type, string value ) : Json( error, type )
{
	if( type == kJSON_NULL )
		this->set_string(value);
	else
		this->m_string = value;
}

JsonValue::~JsonValue()
{
	this->free();
}

void JsonValue::free()
{
	this->m_string.clear();
}

void JsonValue::set_string( string str )
{
	this->free();
	this->m_string	= str;

	int pos = 0;

	// Check if TRUE
	if( this->m_string.compare("true") == 0 )
		Json::set_type(kJSON_TRUE);
	else
	{	// Check if FALSE
		if( this->m_string.compare("false") == 0 )
			Json::set_type(kJSON_FALSE);
		else
		{	// Check if REAL
			pos = 0;
			if( this->m_string.find('.') != string::npos )
				Json::set_type(kJSON_REAL);
			else
			{	// Check if REAL (exponent)
				pos = 0;
				if( this->m_string.find('e') != string::npos )
					Json::set_type(kJSON_REAL);
				else
				{	// Check if INTEGER
					pos = 0;
					if( this->m_string.find_first_of("0123456789") != string::npos )
						Json::set_type(kJSON_INTEGER);
				}
			}
		}
	}
}

/*
* JsonObject class
*
*/
JsonObject::JsonObject( JsonError* error ) : Json(error, kJSON_OBJECT)
{
}

JsonObject::~JsonObject()
{
	this->free();
}

void JsonObject::free()
{
	// Delete the pairs
	map<string,Json*>::iterator it;
	for( it=this->m_keys.begin(); it!=this->m_keys.end(); ++it )
	{
		Json* value = it->second;
		delete value;
	}

	// Delete the vector
	this->m_keys.clear();

	// Call parent
	Json::free();
}

Json* JsonObject::parse( string* s, unsigned int* position )
{
	// Free any previous data
	this->free();

	while( true )
	{
		// Find key
		string key	= this->parse_string(s, position);
		if( key.empty() )
		{
			this->m_error->set_error_code(kJSON_ERR_STRING,*position);
			return NULL;
		}

		// Find :
		unsigned int pos3 = s->find( ':', *position );
		if( pos3 == string::npos )
		{
			this->m_error->set_error_code(kJSON_ERR_COLON, *position);
			return NULL;
		}
		(*position) = pos3+1;

		// Find value
		Json* value = this->parse_value( s, position );
		if( value == NULL )
			return NULL;

		// Create new key
		m_keys[key] = value;

		// Check for end of object or new key/value item
		unsigned int pos = s->find_first_of(",}", *position );
		if( pos == string::npos )
		{
			this->m_error->set_error_code(kJSON_ERR_OBJECT,*position);
			return NULL;
		}
		(*position) = pos+1;

		// End of object?
		if( s->at(pos) == '}' )
			break;
	}

	return this;
}

Json* JsonObject::key_value( string key )
{
	map<string,Json*>::iterator it = this->m_keys.find(key);
	if( it == this->m_keys.end() )
		return NULL;
	else
		return it->second;
}

/*
* JsonArray class
*
*/
JsonArray::JsonArray( JsonError* error ) : Json(error,kJSON_ARRAY)
{
}

JsonArray::~JsonArray()
{
	this->free();
}

void JsonArray::free()
{
	for( unsigned int i=0; i<this->m_values.size(); i++ )
		delete this->m_values.at(i);

	this->m_values.clear();
}

Json* JsonArray::get_at( int index )
{
	if( index < 0 )
		return NULL;

	if( (unsigned int)index >= this->m_values.size() )
		return NULL;

	return this->m_values.at(index);
}

Json* JsonArray::parse( string* s, unsigned int* position )
{
	while( true )
	{
		Json* value = this->parse_value( s, position );
		if( value == NULL )
			return NULL;

		this->m_values.push_back( value );

		int pos = s->find_first_of(",]",*position);
		if( pos == -1 )
		{
			this->m_error->set_error_code( kJSON_ERR_ARRAY, *position );
			return NULL;
		}
		(*position) = pos+1;

		// End of array?
		if( s->at(pos) == ']' )
			break;
	}

	return this;
}

/*
* class JsonError
*
* Class to manage type of errors
*
*/
JsonError::JsonError()
{
	this->m_nCode		= kJSON_ERR_NO_ERROR;
	this->m_nPosition	= 0;
}

void JsonError::set_error_code( JSON_ERROR nCode, int nPosition )
{
	this->m_nCode	= nCode;
	this->m_nPosition	= nPosition;
	switch( this->m_nCode )
	{
		case kJSON_ERR_NO_ERROR		: this->m_sMsg = "No error"; break;
		case kJSON_ERR_STRING		: this->m_sMsg = "String error"; break;
		case kJSON_ERR_COLON		: this->m_sMsg = "Syntax error: missing colon (:)"; break;
		case kJSON_ERR_OBJECT		: this->m_sMsg = "Syntax error: mssing , or } in object"; break;
		case kJSON_ERR_ARRAY		: this->m_sMsg = "Syntax error: missing , or ] in array"; break;
		case kJSON_ERR_PARSE_VALUE	: this->m_sMsg = "Syntax error while parsing value"; break;
		case kJSON_ERR_NO_DATA		: this->m_sMsg = "No data found in string"; break;
		default						:
			{
				char msg[250];
				sprintf( msg, "Error code not found : %02d", this->m_nCode );
				this->m_sMsg = msg;
				break;
			}
	}
}

/*
* json_decode
*
* String to be decodificated
*
*/
Json* json_decode( char* str, JsonError* json_error )
{
	Json* 			root		= NULL;
	unsigned int	position	= 0;
	string			s;

	// Set the string
	s.assign( str );

	while( position < s.length() )
	{
		switch( s[position++] )
		{
			case '{': root = new JsonObject(json_error); break;
			case '[': root = new JsonArray(json_error); break;
		}
		if( root != NULL )
			break;
	}

	if( root != NULL )
	{
		if( root->parse( &s, &position ) == NULL )
		{
			delete root;
			root = NULL;
		}
	}
	else
	{
		json_error->set_error_code(kJSON_ERR_NO_DATA, position);
	}

	return root;
}
```

#### SerialCodes.h
```c
/********************************************************************
 * COPYRIGHT -- Pollux
 ********************************************************************
 * Library: CPP
 * File: SerialCodes.h
 * Author: CEDRIC
 * Created: August 01, 2014
 *******************************************************************/

#include <bur/plctypes.h>
#include <queue>

using namespace std;
typedef queue<string> queue_serial;

// Return the number of serial codes
queue_serial* createSerialQueue();
int getSerialQueueSize( queue_serial* q );
void pushSerialCodeToQueue( queue_serial* q, const char* serial );
const char* popSerialCodeFromQueue(queue_serial* q);
void freeSerialQueue( queue_serial* q);
```

#### SerialCodes.cpp
```cpp
/********************************************************************
 * COPYRIGHT -- Pollux
 ********************************************************************
 * Library: CPP
 * File: SerialCodes.cpp
 * Author: CEDRIC
 * Created: August 01, 2014
 *******************************************************************/

#include <bur/plctypes.h>
#include <queue>
#include <string>
#include "SerialCodes.h"

queue_serial* createSerialQueue()
{
	queue_serial* q = new queue_serial;
	return q;
}

int getSerialQueueSize( queue_serial* q )
{
	int size	= q->size();
	return size;
}

void pushSerialCodeToQueue( queue_serial* q, const char* serial )
{
	string s = serial;
	q->push(s);
}

const char* popSerialCodeFromQueue( queue_serial* q )
{
	string s = q->front();
	q->pop();
	return s.c_str();
}

void freeSerialQueue( queue_serial* q )
{
	delete q;
	q = NULL;
}
```
